FUNCTION_BLOCK ServicesTimingIO EXTENDS SM_ServicesTimingIO
VAR_INPUT
END_VAR
VAR_OUTPUT
END_VAR
VAR
    _testVar_TimingIO : INT;
END_VAR

SUPER^();

// do stuff

//SUPER^();

END_FUNCTION_BLOCK

(* stored: Version 1.1.0.1, ProductVersion 3.1.4018.5
   POU ServicesTimingIO: Id {b0941309-43ee-463d-a122-ae4cf1c5d03b}, SpecialFunc None *)
